// =============================================================================
// FC_FaultHandler
// -----------------------------------------------------------------------------
// PURPOSE:
//   Runs LAST in the FC chain. Overrides the setpoints written by
//   PowerDistribution and ReactiveControl for any inverter that is faulted,
//   lost comms, or in a global stop condition.
//
//   Also writes OperMode to healthy inverters to keep them in Operation and
//   to recover them after a fault or stop.
//
// SIX CONDITIONS HANDLED PER INVERTER:
//
//   A) ForceStop = TRUE (EN_PPC = FALSE in the calling FB)
//      → Stop ALL inverters immediately regardless of health.
//
//   B) Plant_Mode = 2 (FALLBACK)
//      → Stop ALL inverters. Comms to SCADA lost; safe state is zero output.
//
//   C) Individual CommError (partial fault)
//      → Stop only this inverter. Set AnyFault and FaultMask bit.
//      → Inverter's own Modbus watchdog trips it if comms stay down.
//
//   D) Active inverter Error (partial fault, sequence S3.1)
//      → Zero setpoints for this inverter. Set AnyFault and FaultMask bit.
//      → Do not acknowledge while fault is active (ErrClr = 0).
//
//   E) Operator-disabled (Enabled = FALSE, comms healthy, no fault)
//      → HAND BACK TO LOCAL CONTROL: OperMode stays 308, but the control-mode
//        registers switch to manual so the inverter follows its own local HMI
//        setpoints instead of the PPC:
//          WMod   1077 = WCtlMan    (was 1079 WCtlCom)
//          VArMod 1071 = VArCtlMan  (was 303 Off)
//        303 (Off) is wrong here — it releases control and the inverter reverts
//        to MPP tracking. 1079/1072 are wrong too — it would keep following
//        Modbus. Upstream FCs set 1079/303; this FC runs last so these win.
//      → Not a fault: AnyFault and FaultMask are left untouched.
//      → DEPENDS ON FB16: its Modbus write phase must NOT be gated on Enabled,
//        otherwise the mode change is never transmitted and the inverter keeps
//        running under whatever mode it last received.
//
//   F) Healthy inverter (no globalStop, no CommError, no Error)
//      → Write OperMode=308 to keep in Operation (idempotent).
//      → ErrClr one-shot (sequence S3.3): write 26 (Ackn) exactly once
//        when Error transitions 1→0. PrevError array (passed from FB static)
//        tracks previous Error state per inverter for edge detection.
//      → M6 fix: also send ErrClr=26 when Enabled transitions FALSE→TRUE,
//        in case the one-shot fired while the inverter was disabled and the
//        comms block suppressed the write. PrevEnabled tracks Enabled edges.
//      → NOT Available (covers PwrOffReas ≠ 0 OR ELECTRIC_OK = FALSE):
//        InverterMonitor (step ①) computes Available using both conditions.
//        No SkidElectric parameter needed — Available is the single source.
//        Zero setpoints and set AnyFault, but keep OperMode=308 to allow
//        instant recovery once the condition clears. PowerDistribution and
//        ReactiveControl already exclude this inverter via Available; zeroing
//        here is belt-and-suspenders.
//      → DrtStt ≠ 0: inverter is derated (thermal, grid frequency, etc.).
//        Set AnyDerating for HMI alarm. Power is still distributed; WAval
//        already reflects the reduced capacity so the proportional share is
//        naturally lower for a derated unit.
//
// OUTPUTS:
//   AnyFault    — TRUE if any inverter has CommError, Error, or PwrOffReas ≠ 0
//   AnyDerating — TRUE if any healthy inverter has DrtStt ≠ 0
//   FaultMask   — WORD: bit i = inverter i has active CommError or Error
//
// RAMPS RESET:
//   When onlineCount = 0 (all inverters offline), Ramps_Pcmd and Ramps_Qcmd
//   are reset to 0 so both ramps restart from zero when inverters recover.
//
// CALLED FROM: FB_PPC_Controller (step ⑥, last FC in chain)
// =============================================================================

FUNCTION "FC_PPC_FaultHandler" : VOID
{ S7_Optimized_Access := 'TRUE' }
VERSION : 0.1

VAR_INPUT
    // Current plant mode. 2 = FALLBACK → stop all inverters.
    Plant_Mode : INT;

    // TRUE when EN_PPC = FALSE in the calling FB.
    ForceStop : BOOL;
END_VAR

VAR_IN_OUT
    // 10-element inverter array. OperMode, ErrClr and setpoints are written.
    // Available (computed by FC_PPC_InverterMonitor in step ①) is also read here
    // to detect PwrOffReas ≠ 0 / ELECTRIC_OK = FALSE without a separate SkidElectric
    // parameter — InverterMonitor already incorporates those conditions into Available.
    Inverters : Array[0..9] of "Inverter_controller";

    // Reset to 0.0 when all inverters are offline (clean ramp restart).
    Ramps_Pcmd : REAL;

    // Reset to 0.0 when all inverters are offline (clean ramp restart).
    Ramps_Qcmd : REAL;

    // Previous Error state per inverter — stored in FB static section.
    // Used for falling-edge detection to generate the ErrClr one-shot (S3.3).
    PrevError : Array[0..9] of BOOL;

    // Previous Enabled state per inverter — stored in FB static section.
    // Used for rising-edge detection to re-send ErrClr after re-enable (M6).
    PrevEnabled : Array[0..9] of BOOL;
END_VAR

VAR_OUTPUT
    // TRUE if any inverter has an active fault, comms error, or PwrOffReas ≠ 0.
    AnyFault : BOOL;

    // TRUE if any healthy inverter reports a non-zero derating state (DrtStt).
    // Separate from AnyFault — derating does not stop the inverter.
    AnyDerating : BOOL;

    // Bit i = inverter i has active CommError or Error. Used by HMI to show
    // which specific inverters are faulted without browsing all 10 slots.
    FaultMask : WORD;
END_VAR

VAR_TEMP
    i             : INT;    // Loop index
    onlineCount   : INT;    // Inverters fully available after fault evaluation
    globalStop    : BOOL;   // Combined ForceStop / FALLBACK flag
    faultCleared  : BOOL;   // TRUE for one scan when Error transitions 1→0
    enabledRising : BOOL;   // TRUE for one scan when Enabled transitions FALSE→TRUE
END_VAR

BEGIN

    #AnyFault    := FALSE;
    #AnyDerating := FALSE;
    #FaultMask   := WORD#0;
    #onlineCount := 0;

    #globalStop := #ForceStop OR (#Plant_Mode = 2);

    FOR #i := 0 TO 9 DO

        // ── Edge detection ────────────────────────────────────────────────────
        // faultCleared  : Error 1→0 this scan → trigger ErrClr=26 one-shot (S3.3)
        // enabledRising : Enabled FALSE→TRUE → re-send ErrClr=26 in case the
        //   falling-edge one-shot fired while the inverter was disabled (M6 fix)
        #faultCleared  := #PrevError[#i]   AND NOT #Inverters[#i].Error;
        #enabledRising := NOT #PrevEnabled[#i] AND #Inverters[#i].Enabled;
        #PrevError[#i]   := #Inverters[#i].Error;
        #PrevEnabled[#i] := #Inverters[#i].Enabled;

        IF #globalStop THEN
            // ── GLOBAL STOP: issue Stop to ALL inverters (sequence S4) ────────
            // Comms block sees OperMode=303 → writes RemRdy=303 first (S4.1),
            // then InvOpMod=303 (S4.2), satisfying the SMA stop interlock.
            #Inverters[#i].OperMode := 303;   // Stop
            #Inverters[#i].WSpt     := 0;
            #Inverters[#i].VArSpt   := 0;
            #Inverters[#i].PFSpt    := 0;
            #Inverters[#i].WMode    := 303;   // Off
            #Inverters[#i].VArMode  := 303;   // Off
            #Inverters[#i].ErrClr   := 0;

        ELSIF #Inverters[#i].CommError THEN
            // ── INDIVIDUAL COMMS FAULT ────────────────────────────────────────
            // Link broken — write Stop as best-effort. Inverter's own Modbus
            // watchdog will trip it if comms stay down.
            #Inverters[#i].OperMode := 303;
            #Inverters[#i].WSpt     := 0;
            #Inverters[#i].VArSpt   := 0;
            #Inverters[#i].PFSpt    := 0;
            #Inverters[#i].WMode    := 303;
            #Inverters[#i].VArMode  := 303;
            #Inverters[#i].ErrClr   := 0;
            #AnyFault  := TRUE;
            #FaultMask := #FaultMask OR SHL(IN := WORD#1, N := INT_TO_UINT(#i));

        ELSIF #Inverters[#i].Error THEN
            // ── ACTIVE INVERTER FAULT (sequence S3.1) ─────────────────────────
            // ErrStt ≠ 0. Zero setpoints; the inverter trips itself.
            // Do not acknowledge while fault is active (ErrClr = 0).
            // ErrNo (input register 96) should be logged by SCADA (S3.2).
            #Inverters[#i].WSpt    := 0;
            #Inverters[#i].VArSpt  := 0;
            #Inverters[#i].PFSpt   := 0;
            #Inverters[#i].ErrClr  := 0;
            #AnyFault  := TRUE;
            #FaultMask := #FaultMask OR SHL(IN := WORD#1, N := INT_TO_UINT(#i));

        ELSIF NOT #Inverters[#i].Enabled THEN
            // ── OPERATOR-DISABLED — HAND BACK TO LOCAL CONTROL ────────────────
            // [ADDED MOD_DISABLE_PARK]
            // "Disabled" means this inverter is no longer under PPC control — it
            // is handed back to its own local HMI setpoints, not switched off.
            //
            // Mode values matter here (SMA ENUM, Modbus_Comms_Mapping §2.3):
            //   WMod   1077 = WCtlMan   — active power via local HMI
            //   VArMod 1071 = VArCtlMan — reactive power via local HMI
            // NOT 303 (Off), which releases control entirely and lets the
            // inverter revert to MPP tracking, and NOT 1079/1072 (CtlCom),
            // which would keep it following Modbus setpoints.
            //
            // Upstream FCs set these to 1079 / 303; this FC runs last, so the
            // assignments here win.
            //
            // Operator-disable is not a fault — AnyFault / FaultMask untouched.
            #Inverters[#i].OperMode := 308;    // stay in Operation
            #Inverters[#i].WMode    := 1077;   // WCtlMan — local HMI active power
            #Inverters[#i].WSpt     := 0;      // PPC commands nothing
            #Inverters[#i].VArMode  := 1071;   // VArCtlMan — local HMI reactive power
            #Inverters[#i].VArSpt   := 0;
            #Inverters[#i].PFSpt    := 0;
            #Inverters[#i].ErrClr   := 0;

        ELSE
            // ── HEALTHY INVERTER ──────────────────────────────────────────────
            // No globalStop, no CommError, no Error.

            // ErrClr one-shot (sequence S3.3):
            // Write 26 (Ackn) exactly once on:
            //   a) Error falling edge (faultCleared) — normal recovery path
            //   b) Enabled rising edge while Error is clear — re-sends Ackn if
            //      the inverter was disabled when the fault cleared and the
            //      comms block suppressed the one-shot write (M6 fix)
            IF #faultCleared OR (#enabledRising AND NOT #Inverters[#i].Error) THEN
                #Inverters[#i].ErrClr := 26;   // Ackn — one-shot, not continuous
            ELSE
                #Inverters[#i].ErrClr := 0;    // Idle
            END_IF;

            // Keep inverter in Operation (idempotent).
            // Comms block writes RemRdy=308 first (S1.1), then InvOpMod=308 (S1.2).
            #Inverters[#i].OperMode := 308;

            // Derating supervision: DrtStt ≠ 0 means thermal, grid frequency,
            // or other derating is active. WAval already reflects reduced capacity
            // so distribution self-corrects; this flag is purely for HMI visibility.
            IF #Inverters[#i].DrtStt <> 0 THEN
                #AnyDerating := TRUE;
            END_IF;

            // PwrOffReas / ELECTRIC_OK supervision via Available flag:
            //   InverterMonitor (step ①) sets Available = FALSE when
            //   PwrOffReas ≠ 0 OR ELECTRIC_OK = FALSE (switchgear not deliverable).
            //   Since we are already in the ELSE branch (no CommError, no Error),
            //   NOT Available here means exactly that condition.
            // Treat as unavailable: zero setpoints and flag fault.
            // PowerDistribution/ReactiveControl already excluded this inverter
            // via Available; zeroing here is belt-and-suspenders.
            IF NOT #Inverters[#i].Available THEN
                #Inverters[#i].WSpt   := 0;
                #Inverters[#i].VArSpt := 0;
                #Inverters[#i].PFSpt  := 0;
                #AnyFault := TRUE;
                // Not counted — not delivering power
            ELSE
                #onlineCount := #onlineCount + 1;
            END_IF;

        END_IF;

    END_FOR;

    // ── Reset ramps when plant is completely offline ──────────────────────────
    // Ensures both active and reactive ramps restart from zero on recovery
    // rather than jumping to a stale non-zero command.
    IF #onlineCount = 0 THEN
        #Ramps_Pcmd := 0.0;
        #Ramps_Qcmd := 0.0;
    END_IF;

END_FUNCTION
